FUNCTION_BLOCK Fb_Test_init_y
VAR_INPUT
	execute: BOOL;
END_VAR

IF execute  THEN
	MI5.Module2001.Input.SkillInput.SkillInput0.ParameterInput.ParameterInput0.StringValue := 'opc.tcp://192.168.192.118:4840';
	MI5.Module2001.Input.SkillInput.SkillInput0.ParameterInput.ParameterInput1.StringValue := 'MI5.Module1203.Output.PositionSensor';
	MI5.Module2001.Input.SkillInput.SkillInput0.ParameterInput.ParameterInput2.StringValue := 'MI5.Module1203.Input.PositionInput';
	MI5.Module2001.Input.SkillInput.SkillInput0.ParameterInput.ParameterInput3.StringValue := '4';
	MI5.Module2001.Input.SkillInput.SkillInput0.ParameterInput.ParameterInput4.StringValue := 'PLC1';
	MI5.Module2001.Input.SkillInput.SkillInput0.Execute := TRUE;
	IF MI5.Module2001.Output.SkillOutput.SkillOutput0.Done OR MI5.Module2001.Output.SkillOutput.SkillOutput0.Error THEN
		MI5.Module2001.Input.SkillInput.SkillInput0.Execute := FALSE;
		execute := FALSE;
	END_IF
END_IF

END_FUNCTION_BLOCK

(* stored: Version 1.1.0.1, ProductVersion 3.1.0.25
   POU Fb_Test_init_y: Id {3b837eb5-f2ad-411d-b393-a70f629cc15c} *)
